TYPE ST_PNOutput_InputGridControl :
STRUCT
	w_Status					:	WORD;
	w_Warnings					:	WORD;
	w_Faults					:	WORD;
	ui_InputGridStatus			:	UINT;
END_STRUCT
END_TYPE

(* stored: Version 1.1.0.1, ProductVersion 3.1.4026.18
   DUT ST_PNOutput_InputGridControl: Id {9af3bac7-79b2-4e73-ad1b-9a79dba77b9c} *)
